# EPICS substitutions: filter/filter.substitutions
# filter.substitutions

file "$(OPTICS)/opticsApp/Db/filterBladeNoSensor.db" {
  pattern
  {P,      R,        N,   DESC,           OUT                  OUT_STRING,  IN_STRING}
  {BL172:,   filter:,  1,   "Filter 1",     "E1608:Bd1",   "Out",       "In"}
  {BL172:,   filter:,  2,   "Filter 2",     "E1608:Bd2",   "Out",       "In"}
  {BL172:,   filter:,  3,   "Filter 3",     "E1608:Bd3",   "Out",       "In"}
  {BL172:,   filter:,  4,   "Filter 4",     "E1608:Bd4",   "Out",       "In"}
}

file "$(OPTICS)/opticsApp/Db/filterDrive.db" {
  {P="BL172:", R="filter:", DESC="Filters", KEV="BL172:filter:energy_calc"}
}

file "$(OPTICS)/opticsApp/Db/energy_calc.db" {
  {P="BL172:", R="filter:", DESC="Set", angle="IMS:1.RBV",setangle="IMS:1.VAL"
}
